(* Logix 5000 project; controller EuniceF_ICA3 vendor 1 type 14 code 150 rev 37.11; software revision 37.00 *)

TASK MainTask (continuous, watchdog 500 ms) : MainProgram

MODULES
   Local : vendor 1 type 14 code 150 (Compact 0, rev 37.11)
      Discrete_IO : Embedded (Compact 1, rev 3.1, Output RPI 20 ms)
      Analog_IO : Embedded (Compact 2, rev 1.1, Output RPI 80 ms)
      Counters : Embedded (Compact 3, rev 1.1, Output RPI 20 ms)
END_MODULES

VAR_GLOBAL   (* controller tags *)
   FORWARD : ALIAS FOR Local:1:I.Data.13;
   LOCK : BOOL := 1;
   M1 : ALIAS FOR Local:1:O.Data.0;
   M2 : ALIAS FOR Local:1:O.Data.1;
   M3 : ALIAS FOR Local:1:O.Data.2;
   RESET : ALIAS FOR Local:1:I.Data.15;
   REVERSE : ALIAS FOR Local:1:I.Data.14;
   START : ALIAS FOR Local:1:I.Data.11;
   STOP : ALIAS FOR Local:1:I.Data.9;
END_VAR

PROGRAM MainProgram   (* main routine MainRoutine *)

ROUTINE MainRoutine   (* ladder *)
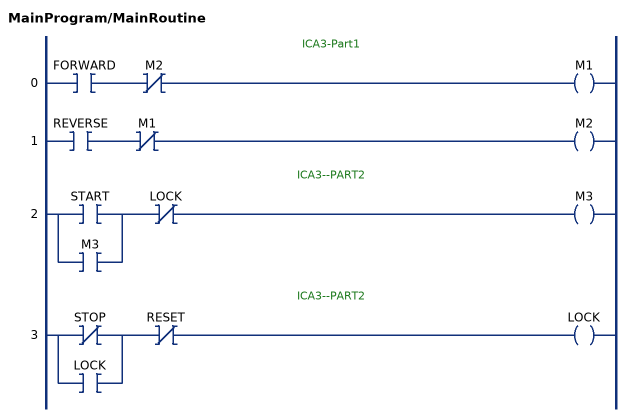
   // ICA3-Part1
   0: XIC(FORWARD)XIO(M2)OTE(M1);
   1: XIC(REVERSE)XIO(M1)OTE(M2);
   // ICA3--PART2
   2: [XIC(START) ,XIC(M3) ]XIO(LOCK)OTE(M3);
   // ICA3--PART2
   3: [XIO(STOP) ,XIC(LOCK) ]XIO(RESET)OTE(LOCK);
END_ROUTINE
END_PROGRAM
